// TIA Portal V15.1 export
// export: Created 2024-06-21T08:40:51.5556217Z, ExportSetting WithDefaults, DisplayName Totally Integrated Automation Portal, DisplayVersion V15.1 Update 5, DisplayName TIA Portal Openness, DisplayVersion V15.1 Update 5, DisplayName SINAMICS Startdrive Advanced, DisplayVersion V15.1, DisplayName G130, G150, S120, S150, SINAMICS MV, S210, DisplayVersion V15.1, DisplayName G110M, G120, G120C, G120D, G120P, DisplayVersion V15.1, DisplayName STEP 7 Professional, DisplayVersion V15.1 Update 5, DisplayName STEP 7 Safety, DisplayVersion V15.1, DisplayName WinCC Professional, DisplayVersion V15.1 Update 5, DisplayName SIMATIC Visualization Architect, DisplayVersion V15.1
FUNCTION_BLOCK "FSafety"   // FB7000, F_FBD
TITLE = FailSafe Program
{ S7_Optimized_Access := 'TRUE' }
VERSION : 0.1
// stored: AutoNumber false, IsIECCheckEnabled false, UDAEnableTagReadback false
BEGIN

REGION Network 1: **** 1 - Inputs **** Safety Signals From PLCyyy / **** 1 - Inputs **** Safety Signals From PLC308
   // Safety Signals From Other PLC
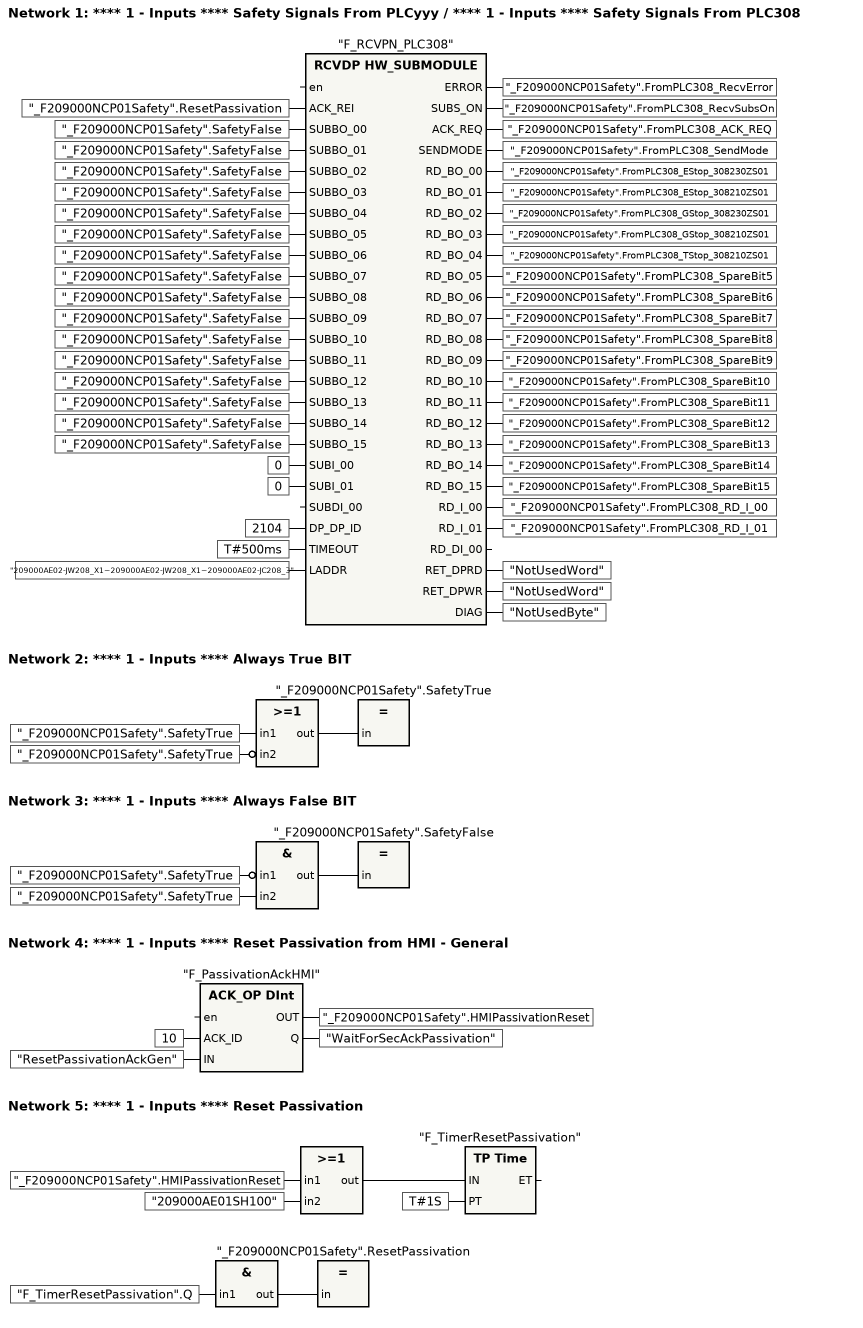
   "F_RCVPN_PLC308"(ACK_REI := "_F209000NCP01Safety".ResetPassivation,   // RCVDP
                    SUBBO_00 := "_F209000NCP01Safety".SafetyFalse,
                    SUBBO_01 := "_F209000NCP01Safety".SafetyFalse,
                    SUBBO_02 := "_F209000NCP01Safety".SafetyFalse,
                    SUBBO_03 := "_F209000NCP01Safety".SafetyFalse,
                    SUBBO_04 := "_F209000NCP01Safety".SafetyFalse,
                    SUBBO_05 := "_F209000NCP01Safety".SafetyFalse,
                    SUBBO_06 := "_F209000NCP01Safety".SafetyFalse,
                    SUBBO_07 := "_F209000NCP01Safety".SafetyFalse,
                    SUBBO_08 := "_F209000NCP01Safety".SafetyFalse,
                    SUBBO_09 := "_F209000NCP01Safety".SafetyFalse,
                    SUBBO_10 := "_F209000NCP01Safety".SafetyFalse,
                    SUBBO_11 := "_F209000NCP01Safety".SafetyFalse,
                    SUBBO_12 := "_F209000NCP01Safety".SafetyFalse,
                    SUBBO_13 := "_F209000NCP01Safety".SafetyFalse,
                    SUBBO_14 := "_F209000NCP01Safety".SafetyFalse,
                    SUBBO_15 := "_F209000NCP01Safety".SafetyFalse,
                    SUBI_00 := 0,
                    SUBI_01 := 0,
                    DP_DP_ID := 2104,
                    TIMEOUT := T#500ms,
                    LADDR := "209000AE02-JW208_X1~209000AE02-JW208_X1~209000AE02-JC208_3",
                    ERROR => "_F209000NCP01Safety".FromPLC308_RecvError,
                    SUBS_ON => "_F209000NCP01Safety".FromPLC308_RecvSubsOn,
                    ACK_REQ => "_F209000NCP01Safety".FromPLC308_ACK_REQ,
                    SENDMODE => "_F209000NCP01Safety".FromPLC308_SendMode,
                    RD_BO_00 => "_F209000NCP01Safety".FromPLC308_EStop_308230ZS01,
                    RD_BO_01 => "_F209000NCP01Safety".FromPLC308_EStop_308210ZS01,
                    RD_BO_02 => "_F209000NCP01Safety".FromPLC308_GStop_308230ZS01,
                    RD_BO_03 => "_F209000NCP01Safety".FromPLC308_GStop_308210ZS01,
                    RD_BO_04 => "_F209000NCP01Safety".FromPLC308_TStop_308210ZS01,
                    RD_BO_05 => "_F209000NCP01Safety".FromPLC308_SpareBit5,
                    RD_BO_06 => "_F209000NCP01Safety".FromPLC308_SpareBit6,
                    RD_BO_07 => "_F209000NCP01Safety".FromPLC308_SpareBit7,
                    RD_BO_08 => "_F209000NCP01Safety".FromPLC308_SpareBit8,
                    RD_BO_09 => "_F209000NCP01Safety".FromPLC308_SpareBit9,
                    RD_BO_10 => "_F209000NCP01Safety".FromPLC308_SpareBit10,
                    RD_BO_11 => "_F209000NCP01Safety".FromPLC308_SpareBit11,
                    RD_BO_12 => "_F209000NCP01Safety".FromPLC308_SpareBit12,
                    RD_BO_13 => "_F209000NCP01Safety".FromPLC308_SpareBit13,
                    RD_BO_14 => "_F209000NCP01Safety".FromPLC308_SpareBit14,
                    RD_BO_15 => "_F209000NCP01Safety".FromPLC308_SpareBit15,
                    RD_I_00 => "_F209000NCP01Safety".FromPLC308_RD_I_00,
                    RD_I_01 => "_F209000NCP01Safety".FromPLC308_RD_I_01,
                    RET_DPRD => "NotUsedWord",
                    RET_DPWR => "NotUsedWord",
                    DIAG => "NotUsedByte");
END_REGION

REGION Network 2: **** 1 - Inputs **** Always True BIT
   // Always True
   "_F209000NCP01Safety".SafetyTrue := "_F209000NCP01Safety".SafetyTrue OR NOT "_F209000NCP01Safety".SafetyTrue;
END_REGION

REGION Network 3: **** 1 - Inputs **** Always False BIT
   // Always False
   "_F209000NCP01Safety".SafetyFalse := NOT "_F209000NCP01Safety".SafetyTrue AND "_F209000NCP01Safety".SafetyTrue;
END_REGION

REGION Network 4: **** 1 - Inputs **** Reset Passivation from HMI - General
   // Reset Passivation from HMI
   "F_PassivationAckHMI"(ACK_ID := 10,   // ACK_OP
                         IN := "ResetPassivationAckGen",
                         OUT => "_F209000NCP01Safety".HMIPassivationReset,
                         Q => "WaitForSecAckPassivation");
END_REGION

REGION Network 5: **** 1 - Inputs **** Reset Passivation
   // General Reset Passivation
   "F_TimerResetPassivation".TP(IN := "_F209000NCP01Safety".HMIPassivationReset OR "209000AE01SH100",
                           PT := T#1S);
   "_F209000NCP01Safety".ResetPassivation := "F_TimerResetPassivation".Q;
END_REGION

REGION Network 6: **** 1 - Inputs **** Emergency Stop Inputs / **** 1 - Inputs **** Safety Inputs
   // Emergency Stop Inputs PLC
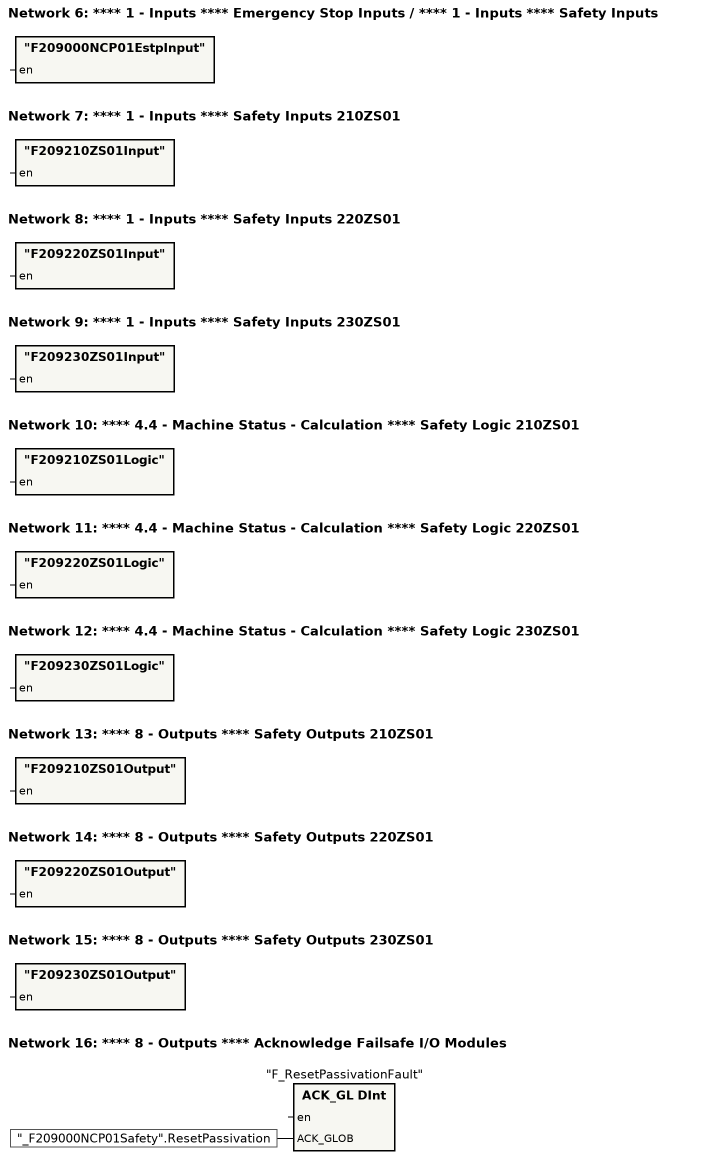
   "F209000NCP01EstpInput"();
END_REGION

REGION Network 7: **** 1 - Inputs **** Safety Inputs 210ZS01
   "F209210ZS01Input"();
END_REGION

REGION Network 8: **** 1 - Inputs **** Safety Inputs 220ZS01
   "F209220ZS01Input"();
END_REGION

REGION Network 9: **** 1 - Inputs **** Safety Inputs 230ZS01
   "F209230ZS01Input"();
END_REGION

REGION Network 10: **** 4.4 - Machine Status - Calculation **** Safety Logic 210ZS01
   "F209210ZS01Logic"();
END_REGION

REGION Network 11: **** 4.4 - Machine Status - Calculation **** Safety Logic 220ZS01
   "F209220ZS01Logic"();
END_REGION

REGION Network 12: **** 4.4 - Machine Status - Calculation **** Safety Logic 230ZS01
   "F209230ZS01Logic"();
END_REGION

REGION Network 13: **** 8 - Outputs **** Safety Outputs 210ZS01
   "F209210ZS01Output"();
END_REGION

REGION Network 14: **** 8 - Outputs **** Safety Outputs 220ZS01
   "F209220ZS01Output"();
END_REGION

REGION Network 15: **** 8 - Outputs **** Safety Outputs 230ZS01
   "F209230ZS01Output"();
END_REGION

REGION Network 16: **** 8 - Outputs **** Acknowledge Failsafe I/O Modules
   // Acknowledge All Failsafe I/O Modules
   "F_ResetPassivationFault"(ACK_GLOB := "_F209000NCP01Safety".ResetPassivation);   // ACK_GL
END_REGION

REGION Network 17: **** 8 - Outputs **** Safety Signals To PLC212
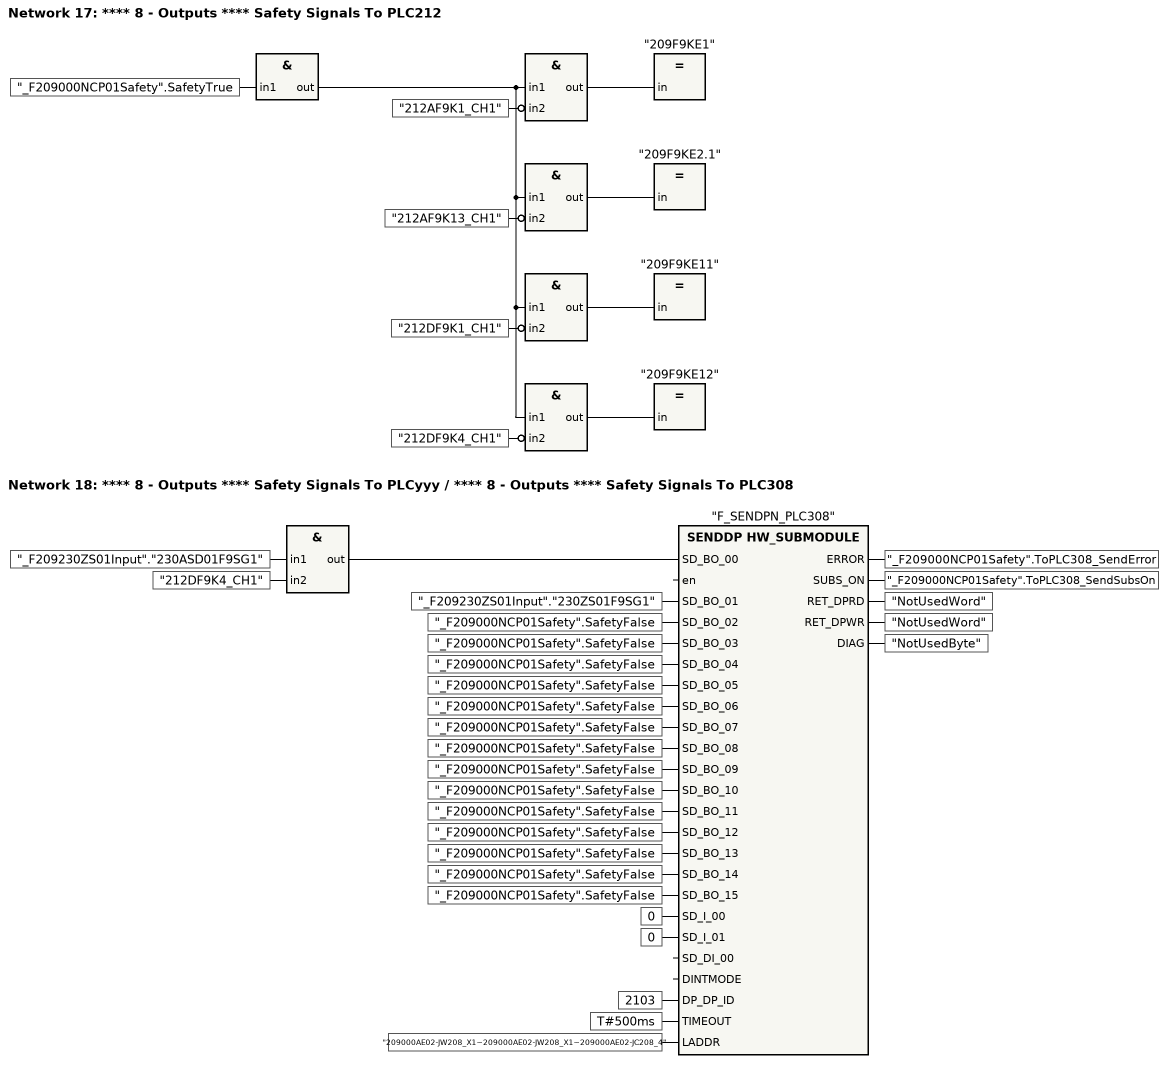
   "209F9KE1" := "_F209000NCP01Safety".SafetyTrue AND NOT "212AF9K1_CH1";
   "209F9KE2.1" := "_F209000NCP01Safety".SafetyTrue AND NOT "212AF9K13_CH1";
   "209F9KE11" := "_F209000NCP01Safety".SafetyTrue AND NOT "212DF9K1_CH1";
   "209F9KE12" := "_F209000NCP01Safety".SafetyTrue AND NOT "212DF9K4_CH1";
END_REGION

REGION Network 18: **** 8 - Outputs **** Safety Signals To PLCyyy / **** 8 - Outputs **** Safety Signals To PLC308
   // Safety Signals To Other PLC
   "F_SENDPN_PLC308"(SD_BO_00 := "_F209230ZS01Input"."230ASD01F9SG1" AND "212DF9K4_CH1",   // SENDDP
                     SD_BO_01 := "_F209230ZS01Input"."230ZS01F9SG1",
                     SD_BO_02 := "_F209000NCP01Safety".SafetyFalse,
                     SD_BO_03 := "_F209000NCP01Safety".SafetyFalse,
                     SD_BO_04 := "_F209000NCP01Safety".SafetyFalse,
                     SD_BO_05 := "_F209000NCP01Safety".SafetyFalse,
                     SD_BO_06 := "_F209000NCP01Safety".SafetyFalse,
                     SD_BO_07 := "_F209000NCP01Safety".SafetyFalse,
                     SD_BO_08 := "_F209000NCP01Safety".SafetyFalse,
                     SD_BO_09 := "_F209000NCP01Safety".SafetyFalse,
                     SD_BO_10 := "_F209000NCP01Safety".SafetyFalse,
                     SD_BO_11 := "_F209000NCP01Safety".SafetyFalse,
                     SD_BO_12 := "_F209000NCP01Safety".SafetyFalse,
                     SD_BO_13 := "_F209000NCP01Safety".SafetyFalse,
                     SD_BO_14 := "_F209000NCP01Safety".SafetyFalse,
                     SD_BO_15 := "_F209000NCP01Safety".SafetyFalse,
                     SD_I_00 := 0,
                     SD_I_01 := 0,
                     DP_DP_ID := 2103,
                     TIMEOUT := T#500ms,
                     LADDR := "209000AE02-JW208_X1~209000AE02-JW208_X1~209000AE02-JC208_4",
                     ERROR => "_F209000NCP01Safety".ToPLC308_SendError,
                     SUBS_ON => "_F209000NCP01Safety".ToPLC308_SendSubsOn,
                     RET_DPRD => "NotUsedWord",
                     RET_DPWR => "NotUsedWord",
                     DIAG => "NotUsedByte");
END_REGION
END_FUNCTION_BLOCK
